FUNCTION_BLOCK LinearSequence EXTENDS ModuleSequenceBase
VAR_INPUT
	i_primitiveIds: ARRAY [ResiConst.ARR_MIN..ResiConst.MODULE_SEQ_ARR_MAX] OF UINT;
	i_primitiveParams: ARRAY [ResiConst.ARR_MIN..ResiConst.MODULE_SEQ_ARR_MAX] OF ParameterSet;
END_VAR
VAR
	i: UINT;
	
	m_sequenceFinished: BOOL;
	m_primitiveId: UINT;
	m_res: EOperationResult;
END_VAR

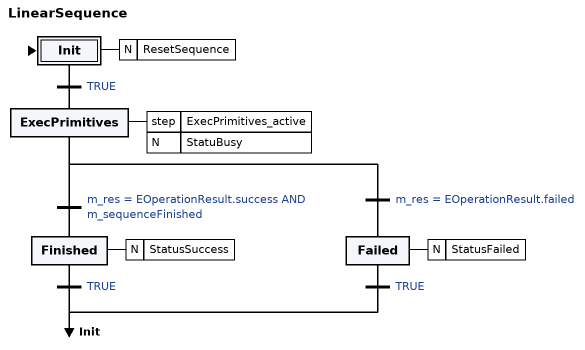
INITIAL_STEP Init:
    ResetSequence(N);
END_STEP
TRANSITION FROM Init TO ExecPrimitives
    := TRUE;
END_TRANSITION
STEP ExecPrimitives:
    ExecPrimitives_active(N);  // step action
    StatuBusy(N);
END_STEP
TRANSITION FROM ExecPrimitives TO Finished
    := m_res = EOperationResult.success AND m_sequenceFinished;
END_TRANSITION
STEP Finished:
    StatusSuccess(N);
END_STEP
TRANSITION FROM Finished TO Init
    := TRUE;
END_TRANSITION
TRANSITION FROM ExecPrimitives TO Failed
    := m_res = EOperationResult.failed;
END_TRANSITION
STEP Failed:
    StatusFailed(N);
END_STEP
TRANSITION FROM Failed TO Init
    := TRUE;
END_TRANSITION

ACTION ExecPrimitives_active:
m_primitiveId := i_primitiveIds[i];

IF m_primitiveId = ESpecialBehaviorIds.empty THEN
	m_sequenceFinished := TRUE;
ELSE
	m_res := m_ptrProcessManager^.Execute(
		i_type := EBehaviorType.control_primitive,
		i_id := m_primitiveId,
		i_params := i_primitiveParams[i]);
		
	IF m_res = EOperationResult.success THEN
		i := i + 1;
	END_IF
END_IF
END_ACTION

PROPERTY Postcondition : IExpression
GET
VAR
	i: UINT;
END_VAR
FOR i := ResiConst.ARR_MIN TO ResiConst.MODULE_SEQ_ARR_MAX DO
	// find the postcondition of the last defined primitive
	IF i_primitiveIds[i] = ESpecialBehaviorIds.empty THEN
		Postcondition := m_ptrProcessManager^.GetBehaviorPtr(EBehaviorType.control_primitive, i_primitiveIds[i - 1])^.Postcondition;
		RETURN;
	END_IF
END_FOR
END_GET
END_PROPERTY

PROPERTY Precondition : IExpression
GET
// precondition of the first defined primitive
Precondition := m_ptrProcessManager^.GetBehaviorPtr(EBehaviorType.control_primitive, i_primitiveIds[ResiConst.ARR_MIN])^.Precondition;
END_GET
END_PROPERTY

METHOD Reset : BOOL
VAR_INPUT
END_VAR
i := ResiConst.ARR_MIN;
m_sequenceFinished := FALSE;
END_METHOD

ACTION ResetSequence:
i := 0;
m_sequenceFinished := FALSE;
m_primitiveId := 0;
o_status := EOperationResult.none;
END_ACTION

ACTION StatuBusy:
o_status := EOperationResult.busy;
END_ACTION

ACTION StatusFailed:
o_status := EOperationResult.failed;
END_ACTION

ACTION StatusSuccess:
o_status := EOperationResult.success;
END_ACTION

END_FUNCTION_BLOCK

(* stored: Version 1.1.0.1
   POU LinearSequence: Id {7bfe67c7-39a5-4041-bd9c-42dee39d3b48}, SpecialFunc None
   Folder Actions: Id {bf14da36-bb7c-4f30-9168-2fa17661aacf}
   Action ExecPrimitives_active: Id {31c24fbe-4b5e-4a19-a139-be1b21f788c7}
   Property Postcondition: Id {b5e893dc-bc1d-433c-8ee9-cb3af9c2c6f4}
   Get Get: Id {4168af93-e3ef-4bb8-bd80-9eab6275e2a4}
   Property Precondition: Id {8e2339c2-4b45-492c-a4ff-6f0e298ee0fe}
   Get Get: Id {528fc167-39ba-45d7-a27a-a3e70ad933ea}
   Method Reset: Id {f6aa9bdd-3471-4d4f-8c10-c0d7dca0437c}
   Action ResetSequence: Id {399dbdc9-980b-4c83-9982-40ce286167b6}
   Action StatuBusy: Id {05cdfa96-4fe8-41c2-8690-174f1709df4a}
   Action StatusFailed: Id {e53780ab-310e-4193-a6c3-0ef3e451769c}
   Action StatusSuccess: Id {04a21b82-0752-4a4a-afd8-d7068cd91112} *)
